TYPE ST_Diagnostics_Recipe :
	STRUCT
		Length				: LREAL;
//		LeftAxis			: ST_AxisRecipe;
//		RightAxis			: ST_AxisRecipe;
		CylinderExtendTime	: LREAL;
		CylinderRetractTime : LREAL;
	END_STRUCT
END_TYPE

(* stored: Version 1.1.0.1, ProductVersion 3.1.4024.15
   DUT ST_Diagnostics_Recipe: Id {41c69f34-a22c-44a0-9f2f-bbb637d49425} *)
